FUNCTION_BLOCK SUBSCRIBE_4 (* Four-variable Subscriber *)
  (* Standard: 61499-2 *)
  (* Version 0.0, 2000-11-27, JHC, Rockwell Automation, Saved for CODEC_TEST *)
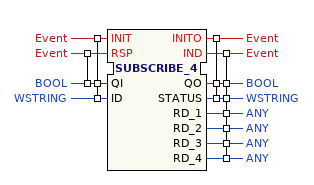
  EVENT_INPUT
    INIT WITH QI, ID; (* Service Initialization *)
    RSP WITH QI; (* Service Response *)
  END_EVENT
  EVENT_OUTPUT
    INITO WITH QO, STATUS; (* Initialization Confirm *)
    IND WITH QO, STATUS, RD_1, RD_2, RD_3, RD_4; (* Service Indication *)
  END_EVENT
  VAR_INPUT
    QI : BOOL; (* Event Input Qualifier *)
    ID : WSTRING; (* Connection Identifier *)
  END_VAR
  VAR_OUTPUT
    QO : BOOL; (* Event Output Qualifier *)
    STATUS : WSTRING; (* Service Status *)
    RD_1 : ANY; (* Subscribed Data *)
    RD_2 : ANY; (* Subscribed Data *)
    RD_3 : ANY; (* Subscribed Data *)
    RD_4 : ANY; (* Subscribed Data *)
  END_VAR
END_FUNCTION_BLOCK
